FUNCTION FC_Percentage_TO_Current4_20Raw : INT
VAR_INPUT
	f : REAL;
END_VAR
VAR
	nIntMax : INT := 32767;
	nIntMin : INT := 6553;
END_VAR

FC_Percentage_TO_Current4_20Raw := REAL_TO_INT(nIntMin + (f/100)*(nIntMax-nIntMin));

END_FUNCTION

(* stored: Version 1.1.0.1, ProductVersion 3.1.4024.0
   POU FC_Percentage_TO_Current4_20Raw: Id {225bd0aa-1131-465c-819c-c641e65bd6ce}, SpecialFunc None *)
